// LS Electric XG5000 project: timer
// PLC LSPLC
// module base 0 slot 0: 입출력 모듈:XBC-DR30S (DC 24V 입력 18점, 릴레이 출력 12점)

PROGRAM timer (task: 스캔 프로그램)

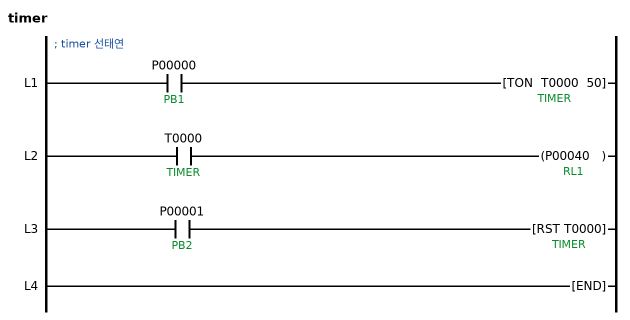
// timer 선태연
; L1
LOAD      P00000	// PB1
TON       T0000 50	// TIMER
; L2
LOAD      T0000	// TIMER
OUT       P00040	// RL1
; L3
LOAD      P00001	// PB2
RST       T0000	// TIMER
; L4
END